{attribute 'qualified_only'}
{attribute 'strict'}
TYPE E_AXIS_CtrlState : (
	IDLE,
	JOG,
	MOVEVELO1,
	MOVEVELO2,
	MOVERELATIVE,
	MOVEABSOLUTE,
	//E_AXIS_HOMINGPOS,
	STOPPOS,
	HALT,
	FASTSTOP
);
END_TYPE

(* stored: Version 1.1.0.1
   DUT E_AXIS_CtrlState: Id {960c727b-077a-4ceb-9933-d411f940a10f} *)
